Universal Robots PolyScope program: d02_amp_off.urp

Program d02_amp_off (installation=default directory=/programs createdIn=5.9.1.1031110 lastSavedIn=5.9.1.1031110 robotSerialNumber=20195501059)
Calibrated DH parameters: a=[0.000146, -0.418764, -0.053981, 0.000058, -0.000023, 0]; d=[0.162545, 37.319448, -206.067439, 168.881546, 0.09955, 0.099464]; alpha=[1.57004, -0.001979, 0.002304, 1.570607, -1.57066, 0]; deltaTheta=[0, -0.174616, -1.258233, 1.432844, -0.000001, 0]
Robot Program (runOnlyOnce=true)
  URCap Gripper (Robotiq_Grippers, Robotiq Inc.) dataModel(position=100.0, force=100.0, speed=100.0, positionInDouble=100.0, forceInDouble=100.0, speedInDouble=100.0, slaveIds=[9], blocking=false)
  MoveL speed 250 mm/s, acceleration 1200 mm/s^2 (useActiveTCP=true) feature=Base
    Waypoint Waypoint (Variable): variable(featureName=d02_amp_sw_p)
    URCap Zero FT Sensor (Robotiq_Copilot, Robotiq Inc.) dataModel(NodeInitializedKey=true, WaitForSteadyWrenchOptionKey=true)
    URCap Force Control (Robotiq_Copilot, Robotiq Inc.) dataModel(NodeInitializedKey=true, force_x=0, force_y=0, force_mx=0, force_my=0, force_mz=0, limit_x_neg=-100, limit_y_neg=-100, limit_z_neg=-100, limit_x_pos=100, limit_y_pos=100, limit_z_pos=100, limit_mx_neg=-20, limit_my_neg=-20, limit_mz_neg=-20, limit_mx_pos=20, limit_my_pos=20, limit_mz_pos=20, ft_control_mx=false, ft_control_my=false, ft_control_mz=false, stiffness_x=100, stiffness_y=100, stiffness_z_position=100, stiffness_mx=100, stiffness_my=100, stiffness_mz=100, force_z=20, ft_control_y=false, ft_control_x=false, TranslatableFeatureKey=1, adaptive_stiffness=true, ft_control_z=true, is_force_control_about_actual_position=true, HackTriggeringContributionIsDefinedMethodKey=true)
      Wait Sleep waitTime=2
    Waypoint Waypoint (Variable): variable(featureName=d02_amp_sw_p)
